FUNCTION_BLOCK CamCurveComp IMPLEMENTS I_CamBuildSequence
VAR
	_State			: UDINT;
	_Front			: I_XtsMover;
	_Rear			: I_XtsMover;
	_Virtual		: I_XtsMover;
	_StartPosition	: LREAL := 0;
	_Speed			: LREAL := 200;
	_Acc			: LREAL := 10_000;
	_Dec			: LREAL := 10_000;
	_Jerk			: LREAL := 100_000;
	_Camming		: ST_Camming;
	_Scaling		: ST_CamScalingData;
	_Offset			: DINT;
	_NumOfRotations : LREAL := 1;
END_VAR

{attribute 'monitoring' := 'call'}
{warning 'Add property implementation'}
PROPERTY Busy : BOOL
GET
END_GET
END_PROPERTY

METHOD CyclicLogic
CASE _State OF
	0:
	10:
		_Virtual.MoveToPosition(Position := _StartPosition);
		NextMinorStep(_State);

	11:
		IF NOT _Virtual.CurrentTask.Busy AND NOT _Virtual.CurrentTask.Error THEN
			NextStep(_State);
		END_IF

	20:
        _Camming.camScaling.MasterOffset := 185;
		_Camming.camIn(Master	  := _Virtual.Axis,
					   Slave	  := _Front.Axis,
					   Execute	  := TRUE,
					   CamTableID := 1,
                       Scaling := _Camming.camScaling );
                       
		IF NOT _Camming.camIn.Busy AND NOT _Camming.camIn.Error THEN
			_Camming.camIn(Master := _Front.Axis, Slave := _Rear.Axis, Execute := FALSE);
			NextMinorStep(_State);
		END_IF
            
     21:
        _Camming.camScaling.MasterOffset := 65;
		_Camming.camIn(Master	  := _Virtual.Axis,
					   Slave	  := _Rear.Axis,
					   Execute	  := TRUE,
					   CamTableID := 1,
                       Scaling := _Camming.camScaling );
                       
		IF NOT _Camming.camIn.Busy AND NOT _Camming.camIn.Error THEN
			_Camming.camIn(Master := _Front.Axis, Slave := _Rear.Axis, Execute := FALSE);
			NextStep(_State);
		END_IF   
        
	30:
		_Virtual.Parameters.Velocity	 := _Speed;
		_Virtual.Parameters.Acceleration := _Acc;
		_Virtual.Parameters.Deceleration := _Dec;
		_Virtual.Parameters.Jerk		 := _Jerk;
		_Virtual.MoveRelative(2122 * _NumOfRotations);
		NextMinorStep(_State);

	31:
		IF NOT _Virtual.CurrentTask.Busy AND NOT _Virtual.CurrentTask.Error THEN
			NextStep(_State);
		END_IF

	40:
		_Camming.camOut(Slave := _Rear.Axis, Execute := TRUE);
		IF NOT _Camming.camOut.Busy AND NOT _Camming.camOut.Error THEN
			_Camming.camOut(Slave := _Rear.Axis, Execute := FALSE);
			NextMinorStep(_State);
		END_IF
            
     41:
		_Camming.camOut(Slave := _Front.Axis, Execute := TRUE);
		IF NOT _Camming.camOut.Busy AND NOT _Camming.camOut.Error THEN
			_Camming.camOut(Slave := _Front.Axis, Execute := FALSE);
			SetStep(_State, 0);
		END_IF   
END_CASE
END_METHOD

PROPERTY FrontMover : I_XtsMover
GET
FrontMover := _Front;
END_GET
SET
_Front := FrontMover;
END_SET
END_PROPERTY

PROPERTY RearMover : I_XtsMover
GET
RearMover := _Rear;
END_GET
SET
_Rear := RearMover;
END_SET
END_PROPERTY

METHOD Reset
_Camming.camIn(Master := _Front.Axis, Slave := _Rear.Axis, Execute := FALSE);
_Virtual.Reset();
SetStep(_State, 0);
END_METHOD

METHOD Start
NextStep(_State);
END_METHOD

{warning 'Add method implementation '}
METHOD Stop
END_METHOD

PROPERTY VirtualMover : I_XtsMover
GET
VirtualMover := _Virtual;
END_GET
SET
_Virtual := VirtualMover;
END_SET
END_PROPERTY

END_FUNCTION_BLOCK

(* stored: Version 1.1.0.1, ProductVersion 3.1.4026.21
   POU CamCurveComp: Id {f937d082-501f-4bd0-8638-3078823e3070}, SpecialFunc None
   Property Busy: Id {c85987ea-864e-45eb-83e1-d64e7cd592ed}
   Get Get: Id {989d4fa8-d781-4c2d-9d59-46aa83b00ec7}
   Method CyclicLogic: Id {d8230271-40ec-4c8b-9f3f-3f30beabce9f}
   Property FrontMover: Id {6b2311db-77e9-4021-b4ee-a30ffe0167d7}
   Get Get: Id {6b52eaff-ca1c-4bcb-93e3-29bdfba8c39b}
   Set Set: Id {69e67626-edff-4071-880a-d99a3df22537}
   Property RearMover: Id {f9583fa8-7946-4415-b86b-846c0a1a2110}
   Get Get: Id {271e5b62-3d30-4eca-a42d-1a7b7e7edef8}
   Set Set: Id {5d60ed20-6809-47b3-b3cc-2642e08a105e}
   Method Reset: Id {65c8728d-94af-4b6e-8c10-86f2a9110128}
   Method Start: Id {b447627a-0911-4eee-b681-628cb242439e}
   Method Stop: Id {7f387c0f-46b5-4121-82a5-0208be847f05}
   Property VirtualMover: Id {91904990-cc87-451e-9e65-01a3947abfde}
   Get Get: Id {5d7c1961-9269-4a4f-b46b-3be1d2e7aabe}
   Set Set: Id {aedeb202-eccb-4247-a7a4-7a7e91fb7e76} *)
